Omron CX-Programmer project NewProject (CX-Programmer 9.70)

# PLC NewPLC1: CP1E E20

## Global symbols (name address type ; comment)
0.01 BOOL  ; stop
0.02 BOOL  ; no pb
0.03 BOOL  ; no pb
100.00 BOOL  ; led
100.01 BOOL  ; led2

## Program NewProgram1 (cyclic task 0)

### Section Section1

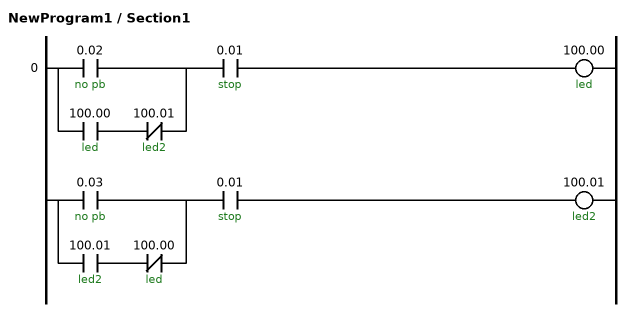
; rung 0
LD 0.02  ; no pb
LD 100.00  ; led
ANDNOT 100.01  ; led2
ORLD
AND 0.01  ; stop
OUT 100.00  ; led
LD 0.03  ; no pb
LD 100.01  ; led2
ANDNOT 100.00  ; led
ORLD
AND 0.01  ; stop
OUT 100.01  ; led2

### Section END
; rung 0
END(001)